(* CODESYS project CodexMonitor.bad.backup.export

Project tree, tasks and I/O mapping:
  visualisation CodexMonitor
*)

// /CodexMonitor
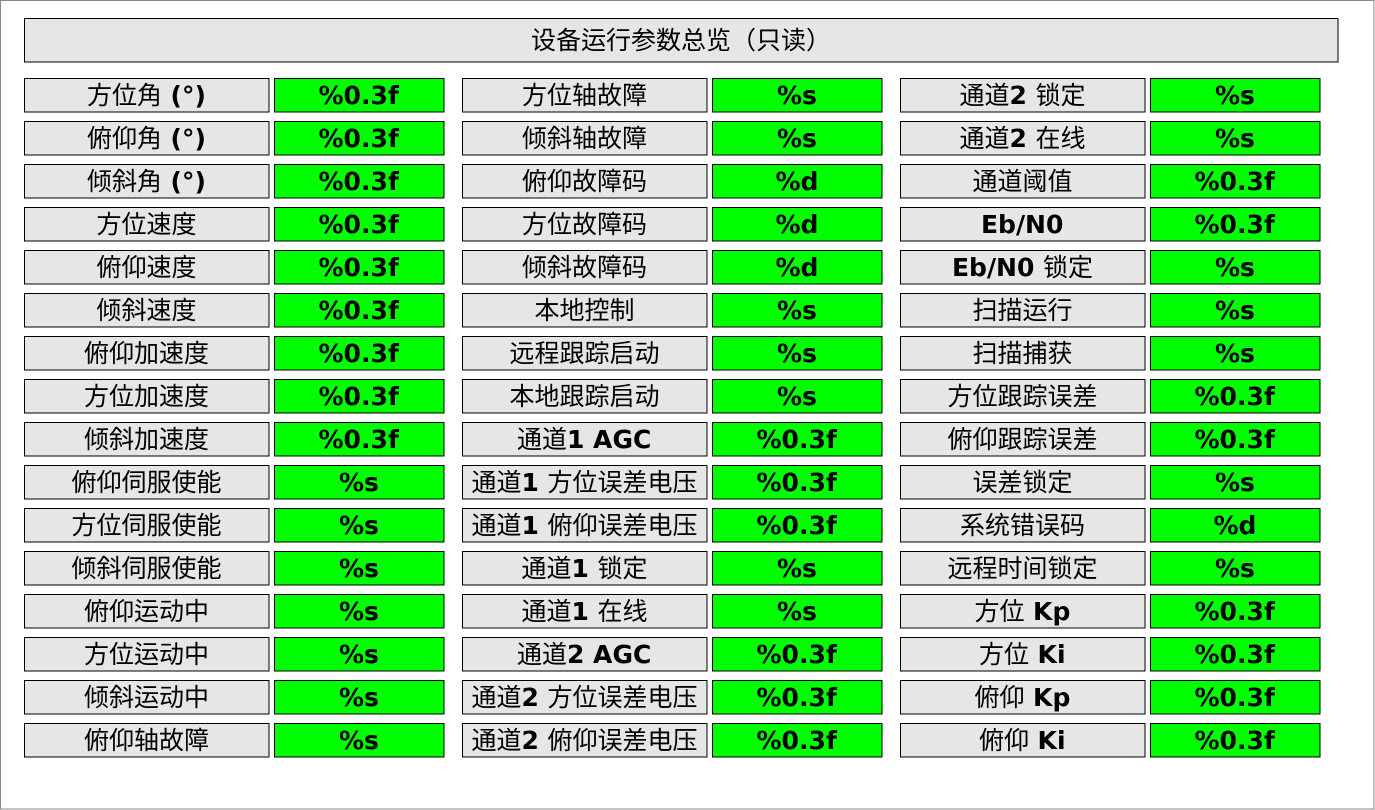
VISUALIZATION CodexMonitor  // 1375x810
    Rectangle (24,18 1314x44), "设备运行参数总览（只读）"
    Rectangle (24,78 245x34), "方位角 (°)"
    Rectangle (274,78 170x34), "%0.3f", text variable: GVL.rFctPosReal_2*(-1)
    Rectangle (24,121 245x34), "俯仰角 (°)"
    Rectangle (274,121 170x34), "%0.3f", text variable: GVL.rFctPosReal_1-90
    Rectangle (24,164 245x34), "倾斜角 (°)"
    Rectangle (274,164 170x34), "%0.3f", text variable: GVL.rFctPosReal_3*(-1)
    Rectangle (24,207 245x34), "方位速度"
    Rectangle (274,207 170x34), "%0.3f", text variable: GVL.rFctVelReal_2*(-1)
    Rectangle (24,250 245x34), "俯仰速度"
    Rectangle (274,250 170x34), "%0.3f", text variable: GVL.rFctVelReal_1
    Rectangle (24,293 245x34), "倾斜速度"
    Rectangle (274,293 170x34), "%0.3f", text variable: GVL.rFctVelReal_3*(-1)
    Rectangle (24,336 245x34), "俯仰加速度"
    Rectangle (274,336 170x34), "%0.3f", text variable: GVL.rFctAccReal_1
    Rectangle (24,379 245x34), "方位加速度"
    Rectangle (274,379 170x34), "%0.3f", text variable: GVL.rFctAccReal_2
    Rectangle (24,422 245x34), "倾斜加速度"
    Rectangle (274,422 170x34), "%0.3f", text variable: GVL.rFctAccReal_3
    Rectangle (24,465 245x34), "俯仰伺服使能"
    Rectangle (274,465 170x34), "%s", text variable: GVL.Axis1Status.bServo_Enable
    Rectangle (24,508 245x34), "方位伺服使能"
    Rectangle (274,508 170x34), "%s", text variable: GVL.Axis2Status.bServo_Enable
    Rectangle (24,551 245x34), "倾斜伺服使能"
    Rectangle (274,551 170x34), "%s", text variable: GVL.Axis3Status.bServo_Enable
    Rectangle (24,594 245x34), "俯仰运动中"
    Rectangle (274,594 170x34), "%s", text variable: GVL.Axis1Status.Moving
    Rectangle (24,637 245x34), "方位运动中"
    Rectangle (274,637 170x34), "%s", text variable: GVL.Axis2Status.Moving
    Rectangle (24,680 245x34), "倾斜运动中"
    Rectangle (274,680 170x34), "%s", text variable: GVL.Axis3Status.Moving
    Rectangle (24,723 245x34), "俯仰轴故障"
    Rectangle (274,723 170x34), "%s", text variable: GVL.Axis1Status.Error
    Rectangle (462,78 245x34), "方位轴故障"
    Rectangle (712,78 170x34), "%s", text variable: GVL.Axis2Status.Error
    Rectangle (462,121 245x34), "倾斜轴故障"
    Rectangle (712,121 170x34), "%s", text variable: GVL.Axis3Status.Error
    Rectangle (462,164 245x34), "俯仰故障码"
    Rectangle (712,164 170x34), "%d", text variable: GVL.Axis1Status.ErrorID
    Rectangle (462,207 245x34), "方位故障码"
    Rectangle (712,207 170x34), "%d", text variable: GVL.Axis2Status.ErrorID
    Rectangle (462,250 245x34), "倾斜故障码"
    Rectangle (712,250 170x34), "%d", text variable: GVL.Axis3Status.ErrorID
    Rectangle (462,293 245x34), "本地控制"
    Rectangle (712,293 170x34), "%s", text variable: GVL.bLocalCtrl
    Rectangle (462,336 245x34), "远程跟踪启动"
    Rectangle (712,336 170x34), "%s", text variable: GVL.bStartTrack
    Rectangle (462,379 245x34), "本地跟踪启动"
    Rectangle (712,379 170x34), "%s", text variable: GVL.bStartLocalAutoTrack
    Rectangle (462,422 245x34), "通道1 AGC"
    Rectangle (712,422 170x34), "%0.3f", text variable: GVL.Chan1AGC
    Rectangle (462,465 245x34), "通道1 方位误差电压"
    Rectangle (712,465 170x34), "%0.3f", text variable: GVL.Chan1Ua
    Rectangle (462,508 245x34), "通道1 俯仰误差电压"
    Rectangle (712,508 170x34), "%0.3f", text variable: GVL.Chan1Ue
    Rectangle (462,551 245x34), "通道1 锁定"
    Rectangle (712,551 170x34), "%s", text variable: GVL.Chan1Lock
    Rectangle (462,594 245x34), "通道1 在线"
    Rectangle (712,594 170x34), "%s", text variable: GVL.Chan1Online
    Rectangle (462,637 245x34), "通道2 AGC"
    Rectangle (712,637 170x34), "%0.3f", text variable: GVL.Chan2AGC
    Rectangle (462,680 245x34), "通道2 方位误差电压"
    Rectangle (712,680 170x34), "%0.3f", text variable: GVL.Chan2Ua
    Rectangle (462,723 245x34), "通道2 俯仰误差电压"
    Rectangle (712,723 170x34), "%0.3f", text variable: GVL.Chan2Ue
    Rectangle (900,78 245x34), "通道2 锁定"
    Rectangle (1150,78 170x34), "%s", text variable: GVL.Chan2Lock
    Rectangle (900,121 245x34), "通道2 在线"
    Rectangle (1150,121 170x34), "%s", text variable: GVL.Chan2Online
    Rectangle (900,164 245x34), "通道阈值"
    Rectangle (1150,164 170x34), "%0.3f", text variable: GVL.Chanthreshold
    Rectangle (900,207 245x34), "Eb/N0"
    Rectangle (1150,207 170x34), "%0.3f", text variable: READ_485.Chan1EB_N0
    Rectangle (900,250 245x34), "Eb/N0 锁定"
    Rectangle (1150,250 170x34), "%s", text variable: READ_485.bEBN0Lock
    Rectangle (900,293 245x34), "扫描运行"
    Rectangle (1150,293 170x34), "%s", text variable: SecurityCheck.bScanRun
    Rectangle (900,336 245x34), "扫描捕获"
    Rectangle (1150,336 170x34), "%s", text variable: SecurityCheck.bScanFound
    Rectangle (900,379 245x34), "方位跟踪误差"
    Rectangle (1150,379 170x34), "%0.3f", text variable: SecurityCheck.AzError
    Rectangle (900,422 245x34), "俯仰跟踪误差"
    Rectangle (1150,422 170x34), "%0.3f", text variable: SecurityCheck.ElError
    Rectangle (900,465 245x34), "误差锁定"
    Rectangle (1150,465 170x34), "%s", text variable: SecurityCheck.bErrorLock
    Rectangle (900,508 245x34), "系统错误码"
    Rectangle (1150,508 170x34), "%d", text variable: GVL.Error_code
    Rectangle (900,551 245x34), "远程时间锁定"
    Rectangle (1150,551 170x34), "%s", text variable: GVL.bRemoteTimeLock
    Rectangle (900,594 245x34), "方位 Kp"
    Rectangle (1150,594 170x34), "%0.3f", text variable: GVL.rvAzKpBase
    Rectangle (900,637 245x34), "方位 Ki"
    Rectangle (1150,637 170x34), "%0.3f", text variable: GVL.rvAzKiBase
    Rectangle (900,680 245x34), "俯仰 Kp"
    Rectangle (1150,680 170x34), "%0.3f", text variable: GVL.rvElKpBase
    Rectangle (900,723 245x34), "俯仰 Ki"
    Rectangle (1150,723 170x34), "%0.3f", text variable: GVL.rvElKiBase
END_VISUALIZATION
